KUKA KRL program: cuadrado.src, cuadrado.dat

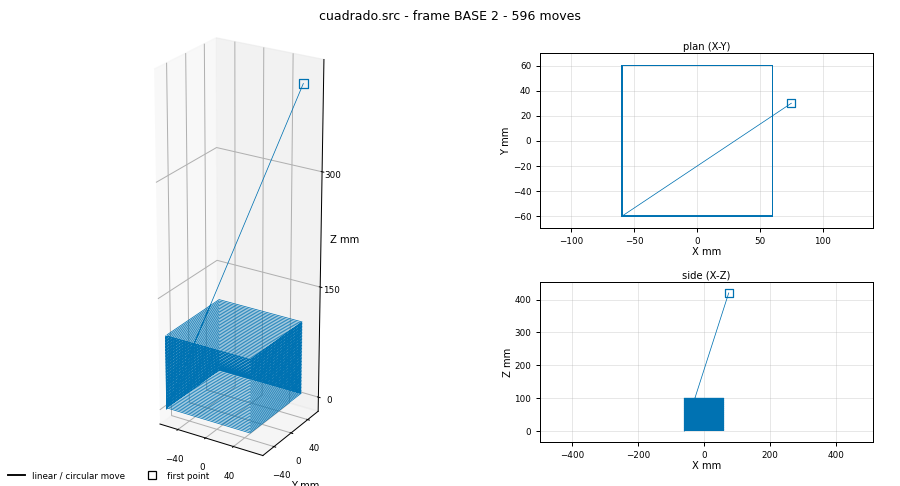
[picture p0: tool path of cuadrado.src in frame BASE 2, 596 of 598 moves have a stored position in this frame; points joined in program order, loops and branches not executed]
--- cuadrado.src ---
&ACCESS RVP
&PARAM TEMPLATE = C:\KRC\Roboter\Template\vorgabe
&PARAM EDITMASK = *
DEF cuadrado( )
;FOLD INI;%{PE}%V3.2.0,%MKUKATPBASIS,%CINIT,%VCOMMON,%P
;FOLD BAS INI;%{E}%V3.2.0,%MKUKATPBASIS,%CINIT,%VINIT,%P
GLOBAL INTERRUPT DECL 3 WHEN $STOPMESS==TRUE DO IR_STOPM ( )
INTERRUPT ON 3
BAS (#INITMOV,0 )
;ENDFOLD (BAS INI)
;FOLD A20 INI;%{E}%V3.2.0,%MKUKATPA20,%CINIT,%VINIT,%P
IF ARC20==TRUE THEN
A20 (ARC_INI)
INTERRUPT DECL 6 WHEN $CYCFLAG[3]==FALSE DO A20(TECH_STOP2)
ENDIF
;ENDFOLD (A20 INI)
;FOLD A10 INI;%{E}%V3.2.0,%MKUKATPARC,%CINIT,%VINIT,%P
IF A10_OPTION==#ACTIVE THEN
INTERRUPT DECL 4 WHEN $CYCFLAG[2]==FALSE DO A10 (#APPL_ERROR)
INTERRUPT DECL 7 WHEN A_ARC_SWI==#ACTIVE DO A10 (#ARC_SEAM)
INTERRUPT DECL 5 WHEN A_FLY_ARC==TRUE DO A10 (#HPU_ARC)
INTERRUPT  ON 5
A10_INI ( )
ENDIF
;ENDFOLD (A10 INI)
;FOLD GRIPPER INI;%{E}%V3.2.0,%MKUKATPGRIPPER,%CINIT,%VINIT,%P
USER_GRP(0,DUMMY,DUMMY,GDEFAULT)
;ENDFOLD (GRIPPER INI)
;FOLD SPOT INI;%{E}%V3.2.0,%MKUKATPSPOT,%CINIT,%VINIT,%P
USERSPOT(#INIT)
;ENDFOLD (SPOT INI)
;FOLD TOUCHSENSE INI;%{E}%V3.2.0,%MKUKATPTS,%CINIT,%VINIT,%P
IF H70_OPTION THEN
INTERRUPT DECL 15 WHEN $MEAS_PULSE[TOUCH_I[TOUCH_ACTIVE].IN_NR] DO H70 (6,CD0 )
INTERRUPT DECL 16 WHEN $ZERO_MOVE DO H70 (7,CD0 )
INTERRUPT DECL 17 WHEN $TECHPAR_C[FG_TOUCH,8]>0.5 DO H70 (8,CD0)
H70 (1,CD0 )
ENDIF
;ENDFOLD (TOUCHSENSE INI)
;FOLD USER INI;%{E}%V3.2.0,%MKUKATPUSER,%CINIT,%VINIT,%P
;Make your modifications here
;ENDFOLD (USER INI)
;ENDFOLD (INI)
; SPEED PTP FOR AXIS
$VEL_AXIS[1] = 15
$VEL_AXIS[2] = 15
$VEL_AXIS[3] = 15
$VEL_AXIS[4] = 15
$VEL_AXIS[5] = 15
$VEL_AXIS[6] = 15
;SMOOTHNESS
$APO.CDIS = 2
;ADVANCE
$ADVANCE = 3
;SET TOOL AND BASE
$TOOL = TOOL_DATA[3]
$BASE = BASE_DATA[2]
;HOME
;FOLD PTP HOME Vel=10% DEFAULT
$BWDSTART=FALSE
$H_POS=XHOME
PDAT_ACT=PDEFAULT
FDAT_ACT=FHOME
BAS(#PTP_DAT )
BAS (#VEL_PTP,10 )
PTP XHOME
;ENDFOLD
;USER PROGRAM
;SPEED $VEL.CP
$VEL.CP=0.025
; OUT[TEMP] = 200
; OUT[vent] = 1
; OUT[RPM] = 25
$OUT[1] = TRUE
WAIT SEC 20
$OUT[1] = FALSE
; USER POSES CALLS
PTP {X 75, Y 30, Z 420, A 0, B 90, C 0}
; USER POSES CALLS
LIN {X -60.0, Y -60.0, Z 0.0, A 0, B 90, C 0} C_DIS
WAIT SEC 3
LIN {X -60.0, Y -60.0, Z 2.0, A 0, B 90, C 0} C_DIS
$OUT[1] = TRUE
WAIT SEC 0.8
LIN {X -60.0, Y -60.0, Z 2.0, A 0, B 90, C 0} C_DIS
LIN {X -60.0, Y -60.0, Z 2.0, A 0, B 90, C 0} C_DIS
LIN {X 60.0, Y -60.0, Z 2.0, A 0, B 90, C 0} C_DIS
LIN {X 60.0, Y 60.0, Z 2.0, A 0, B 90, C 0} C_DIS
LIN {X -60.0, Y 60.0, Z 2.0, A 0, B 90, C 0} C_DIS
LIN {X -60.0, Y -56.5, Z 2.0, A 0, B 90, C 0} C_DIS
$OUT[1] = FALSE

; END LAYER 0
LIN {X -60.0, Y -60.0, Z 2.0, A 0, B 90, C 0} C_DIS
WAIT SEC 3
LIN {X -60.0, Y -60.0, Z 4.0, A 0, B 90, C 0} C_DIS
$OUT[1] = TRUE
WAIT SEC 0.8
LIN {X -60.0, Y -60.0, Z 4.0, A 0, B 90, C 0} C_DIS
LIN {X -60.0, Y -60.0, Z 4.0, A 0, B 90, C 0} C_DIS
LIN {X 57.6, Y -60.0, Z 4.0, A 0, B 90, C 0} C_DIS
LIN {X 60.0, Y -60.0, Z 4.0, A 0, B 90, C 0} C_DIS
LIN {X 60.0, Y 57.6, Z 4.0, A 0, B 90, C 0} C_DIS
LIN {X 60.0, Y 60.0, Z 4.0, A 0, B 90, C 0} C_DIS
LIN {X -57.6, Y 60.0, Z 4.0, A 0, B 90, C 0} C_DIS
LIN {X -60.0, Y 60.0, Z 4.0, A 0, B 90, C 0} C_DIS
LIN {X -60.0, Y -57.6, Z 4.0, A 0, B 90, C 0} C_DIS
$OUT[1] = FALSE

; END LAYER 1
LIN {X -60.0, Y -60.0, Z 4.0, A 0, B 90, C 0} C_DIS
WAIT SEC 3
LIN {X -60.0, Y -60.0, Z 6.0, A 0, B 90, C 0} C_DIS
$OUT[1] = TRUE
WAIT SEC 0.8
LIN {X -60.0, Y -60.0, Z 6.0, A 0, B 90, C 0} C_DIS
LIN {X -60.0, Y -60.0, Z 6.0, A 0, B 90, C 0} C_DIS
LIN {X 55.2, Y -60.0, Z 6.0, A 0, B 90, C 0} C_DIS
LIN {X 60.0, Y -60.0, Z 6.0, A 0, B 90, C 0} C_DIS
LIN {X 60.0, Y 55.2, Z 6.0, A 0, B 90, C 0} C_DIS
LIN {X 60.0, Y 60.0, Z 6.0, A 0, B 90, C 0} C_DIS
LIN {X -55.2, Y 60.0, Z 6.0, A 0, B 90, C 0} C_DIS
LIN {X -60.0, Y 60.0, Z 6.0, A 0, B 90, C 0} C_DIS
LIN {X -60.0, Y -55.2, Z 6.0, A 0, B 90, C 0} C_DIS
LIN {X -60.0, Y -56.5, Z 6.0, A 0, B 90, C 0} C_DIS
$OUT[1] = FALSE

; END LAYER 2
LIN {X -60.0, Y -60.0, Z 6.0, A 0, B 90, C 0} C_DIS
WAIT SEC 3
LIN {X -60.0, Y -60.0, Z 8.0, A 0, B 90, C 0} C_DIS
$OUT[1] = TRUE
WAIT SEC 0.8
LIN {X -60.0, Y -60.0, Z 8.0, A 0, B 90, C 0} C_DIS
LIN {X -60.0, Y -60.0, Z 8.0, A 0, B 90, C 0} C_DIS
LIN {X 52.8, Y -60.0, Z 8.0, A 0, B 90, C 0} C_DIS
LIN {X 60.0, Y -60.0, Z 8.0, A 0, B 90, C 0} C_DIS
LIN {X 60.0, Y 52.8, Z 8.0, A 0, B 90, C 0} C_DIS
LIN {X 60.0, Y 60.0, Z 8.0, A 0, B 90, C 0} C_DIS
LIN {X -52.8, Y 60.0, Z 8.0, A 0, B 90, C 0} C_DIS
LIN {X -60.0, Y 60.0, Z 8.0, A 0, B 90, C 0} C_DIS
LIN {X -60.0, Y -52.8, Z 8.0, A 0, B 90, C 0} C_DIS
LIN {X -60.0, Y -56.5, Z 8.0, A 0, B 90, C 0} C_DIS
$OUT[1] = FALSE

; END LAYER 3
LIN {X -60.0, Y -60.0, Z 8.0, A 0, B 90, C 0} C_DIS
WAIT SEC 3
LIN {X -60.0, Y -60.0, Z 10.0, A 0, B 90, C 0} C_DIS
$OUT[1] = TRUE
WAIT SEC 0.8
LIN {X -60.0, Y -60.0, Z 10.0, A 0, B 90, C 0} C_DIS
LIN {X -60.0, Y -60.0, Z 10.0, A 0, B 90, C 0} C_DIS
LIN {X 50.4, Y -60.0, Z 10.0, A 0, B 90, C 0} C_DIS
LIN {X 60.0, Y -60.0, Z 10.0, A 0, B 90, C 0} C_DIS
LIN {X 60.0, Y 50.4, Z 10.0, A 0, B 90, C 0} C_DIS
LIN {X 60.0, Y 60.0, Z 10.0, A 0, B 90, C 0} C_DIS
LIN {X -50.4, Y 60.0, Z 10.0, A 0, B 90, C 0} C_DIS
LIN {X -60.0, Y 60.0, Z 10.0, A 0, B 90, C 0} C_DIS
LIN {X -60.0, Y -50.4, Z 10.0, A 0, B 90, C 0} C_DIS
LIN {X -60.0, Y -56.5, Z 10.0, A 0, B 90, C 0} C_DIS
$OUT[1] = FALSE

; END LAYER 4
LIN {X -60.0, Y -60.0, Z 10.0, A 0, B 90, C 0} C_DIS
WAIT SEC 3
LIN {X -60.0, Y -60.0, Z 12.0, A 0, B 90, C 0} C_DIS
$OUT[1] = TRUE
WAIT SEC 0.8
LIN {X -60.0, Y -60.0, Z 12.0, A 0, B 90, C 0} C_DIS
LIN {X -60.0, Y -60.0, Z 12.0, A 0, B 90, C 0} C_DIS
LIN {X 48.0, Y -60.0, Z 12.0, A 0, B 90, C 0} C_DIS
LIN {X 60.0, Y -60.0, Z 12.0, A 0, B 90, C 0} C_DIS
LIN {X 60.0, Y 48.0, Z 12.0, A 0, B 90, C 0} C_DIS
LIN {X 60.0, Y 60.0, Z 12.0, A 0, B 90, C 0} C_DIS
LIN {X -48.0, Y 60.0, Z 12.0, A 0, B 90, C 0} C_DIS
LIN {X -60.0, Y 60.0, Z 12.0, A 0, B 90, C 0} C_DIS
LIN {X -60.0, Y -48.0, Z 12.0, A 0, B 90, C 0} C_DIS
LIN {X -60.0, Y -56.5, Z 12.0, A 0, B 90, C 0} C_DIS
$OUT[1] = FALSE

; END LAYER 5
LIN {X -60.0, Y -60.0, Z 12.0, A 0, B 90, C 0} C_DIS
WAIT SEC 3
LIN {X -60.0, Y -60.0, Z 14.0, A 0, B 90, C 0} C_DIS
$OUT[1] = TRUE
WAIT SEC 0.8
LIN {X -60.0, Y -60.0, Z 14.0, A 0, B 90, C 0} C_DIS
LIN {X -60.0, Y -60.0, Z 14.0, A 0, B 90, C 0} C_DIS
LIN {X 45.6, Y -60.0, Z 14.0, A 0, B 90, C 0} C_DIS
LIN {X 60.0, Y -60.0, Z 14.0, A 0, B 90, C 0} C_DIS
LIN {X 60.0, Y 45.6, Z 14.0, A 0, B 90, C 0} C_DIS
LIN {X 60.0, Y 60.0, Z 14.0, A 0, B 90, C 0} C_DIS
LIN {X -45.6, Y 60.0, Z 14.0, A 0, B 90, C 0} C_DIS
LIN {X -60.0, Y 60.0, Z 14.0, A 0, B 90, C 0} C_DIS
LIN {X -60.0, Y -45.6, Z 14.0, A 0, B 90, C 0} C_DIS
LIN {X -60.0, Y -56.5, Z 14.0, A 0, B 90, C 0} C_DIS
$OUT[1] = FALSE

; END LAYER 6
LIN {X -60.0, Y -60.0, Z 14.0, A 0, B 90, C 0} C_DIS
WAIT SEC 3
LIN {X -60.0, Y -60.0, Z 16.0, A 0, B 90, C 0} C_DIS
$OUT[1] = TRUE
WAIT SEC 0.8
LIN {X -60.0, Y -60.0, Z 16.0, A 0, B 90, C 0} C_DIS
LIN {X -60.0, Y -60.0, Z 16.0, A 0, B 90, C 0} C_DIS
LIN {X 43.2, Y -60.0, Z 16.0, A 0, B 90, C 0} C_DIS
LIN {X 60.0, Y -60.0, Z 16.0, A 0, B 90, C 0} C_DIS
LIN {X 60.0, Y 43.2, Z 16.0, A 0, B 90, C 0} C_DIS
LIN {X 60.0, Y 60.0, Z 16.0, A 0, B 90, C 0} C_DIS
LIN {X -43.2, Y 60.0, Z 16.0, A 0, B 90, C 0} C_DIS
LIN {X -60.0, Y 60.0, Z 16.0, A 0, B 90, C 0} C_DIS
LIN {X -60.0, Y -43.2, Z 16.0, A 0, B 90, C 0} C_DIS
LIN {X -60.0, Y -56.5, Z 16.0, A 0, B 90, C 0} C_DIS
$OUT[1] = FALSE

; END LAYER 7
LIN {X -60.0, Y -60.0, Z 16.0, A 0, B 90, C 0} C_DIS
WAIT SEC 3
LIN {X -60.0, Y -60.0, Z 18.0, A 0, B 90, C 0} C_DIS
$OUT[1] = TRUE
WAIT SEC 0.8
LIN {X -60.0, Y -60.0, Z 18.0, A 0, B 90, C 0} C_DIS
LIN {X -60.0, Y -60.0, Z 18.0, A 0, B 90, C 0} C_DIS
LIN {X 40.8, Y -60.0, Z 18.0, A 0, B 90, C 0} C_DIS
LIN {X 60.0, Y -60.0, Z 18.0, A 0, B 90, C 0} C_DIS
LIN {X 60.0, Y 40.8, Z 18.0, A 0, B 90, C 0} C_DIS
LIN {X 60.0, Y 60.0, Z 18.0, A 0, B 90, C 0} C_DIS
LIN {X -40.8, Y 60.0, Z 18.0, A 0, B 90, C 0} C_DIS
LIN {X -60.0, Y 60.0, Z 18.0, A 0, B 90, C 0} C_DIS
LIN {X -60.0, Y -40.8, Z 18.0, A 0, B 90, C 0} C_DIS
LIN {X -60.0, Y -56.5, Z 18.0, A 0, B 90, C 0} C_DIS
$OUT[1] = FALSE

; END LAYER 8
LIN {X -60.0, Y -60.0, Z 18.0, A 0, B 90, C 0} C_DIS
WAIT SEC 3
LIN {X -60.0, Y -60.0, Z 20.0, A 0, B 90, C 0} C_DIS
$OUT[1] = TRUE
WAIT SEC 0.8
LIN {X -60.0, Y -60.0, Z 20.0, A 0, B 90, C 0} C_DIS
LIN {X -60.0, Y -60.0, Z 20.0, A 0, B 90, C 0} C_DIS
LIN {X 38.4, Y -60.0, Z 20.0, A 0, B 90, C 0} C_DIS
LIN {X 60.0, Y -60.0, Z 20.0, A 0, B 90, C 0} C_DIS
LIN {X 60.0, Y 38.4, Z 20.0, A 0, B 90, C 0} C_DIS
LIN {X 60.0, Y 60.0, Z 20.0, A 0, B 90, C 0} C_DIS
LIN {X -38.4, Y 60.0, Z 20.0, A 0, B 90, C 0} C_DIS
LIN {X -60.0, Y 60.0, Z 20.0, A 0, B 90, C 0} C_DIS
LIN {X -60.0, Y -38.4, Z 20.0, A 0, B 90, C 0} C_DIS
LIN {X -60.0, Y -56.5, Z 20.0, A 0, B 90, C 0} C_DIS
$OUT[1] = FALSE

; END LAYER 9
LIN {X -60.0, Y -60.0, Z 20.0, A 0, B 90, C 0} C_DIS
WAIT SEC 3
LIN {X -60.0, Y -60.0, Z 22.0, A 0, B 90, C 0} C_DIS
$OUT[1] = TRUE
WAIT SEC 0.8
LIN {X -60.0, Y -60.0, Z 22.0, A 0, B 90, C 0} C_DIS
LIN {X -60.0, Y -60.0, Z 22.0, A 0, B 90, C 0} C_DIS
LIN {X 36.0, Y -60.0, Z 22.0, A 0, B 90, C 0} C_DIS
LIN {X 60.0, Y -60.0, Z 22.0, A 0, B 90, C 0} C_DIS
LIN {X 60.0, Y 36.0, Z 22.0, A 0, B 90, C 0} C_DIS
LIN {X 60.0, Y 60.0, Z 22.0, A 0, B 90, C 0} C_DIS
LIN {X -36.0, Y 60.0, Z 22.0, A 0, B 90, C 0} C_DIS
LIN {X -60.0, Y 60.0, Z 22.0, A 0, B 90, C 0} C_DIS
LIN {X -60.0, Y -36.0, Z 22.0, A 0, B 90, C 0} C_DIS
LIN {X -60.0, Y -56.5, Z 22.0, A 0, B 90, C 0} C_DIS
$OUT[1] = FALSE

; END LAYER 10
LIN {X -60.0, Y -60.0, Z 22.0, A 0, B 90, C 0} C_DIS
WAIT SEC 3
LIN {X -60.0, Y -60.0, Z 24.0, A 0, B 90, C 0} C_DIS
$OUT[1] = TRUE
WAIT SEC 0.8
LIN {X -60.0, Y -60.0, Z 24.0, A 0, B 90, C 0} C_DIS
LIN {X -60.0, Y -60.0, Z 24.0, A 0, B 90, C 0} C_DIS
LIN {X 33.6, Y -60.0, Z 24.0, A 0, B 90, C 0} C_DIS
LIN {X 60.0, Y -60.0, Z 24.0, A 0, B 90, C 0} C_DIS
LIN {X 60.0, Y 33.6, Z 24.0, A 0, B 90, C 0} C_DIS
LIN {X 60.0, Y 60.0, Z 24.0, A 0, B 90, C 0} C_DIS
LIN {X -33.6, Y 60.0, Z 24.0, A 0, B 90, C 0} C_DIS
LIN {X -60.0, Y 60.0, Z 24.0, A 0, B 90, C 0} C_DIS
LIN {X -60.0, Y -33.6, Z 24.0, A 0, B 90, C 0} C_DIS
LIN {X -60.0, Y -56.5, Z 24.0, A 0, B 90, C 0} C_DIS
$OUT[1] = FALSE

; END LAYER 11
LIN {X -60.0, Y -60.0, Z 24.0, A 0, B 90, C 0} C_DIS
WAIT SEC 3
LIN {X -60.0, Y -60.0, Z 26.0, A 0, B 90, C 0} C_DIS
$OUT[1] = TRUE
WAIT SEC 0.8
LIN {X -60.0, Y -60.0, Z 26.0, A 0, B 90, C 0} C_DIS
LIN {X -60.0, Y -60.0, Z 26.0, A 0, B 90, C 0} C_DIS
LIN {X 31.2, Y -60.0, Z 26.0, A 0, B 90, C 0} C_DIS
LIN {X 60.0, Y -60.0, Z 26.0, A 0, B 90, C 0} C_DIS
LIN {X 60.0, Y 31.2, Z 26.0, A 0, B 90, C 0} C_DIS
LIN {X 60.0, Y 60.0, Z 26.0, A 0, B 90, C 0} C_DIS
LIN {X -31.2, Y 60.0, Z 26.0, A 0, B 90, C 0} C_DIS
LIN {X -60.0, Y 60.0, Z 26.0, A 0, B 90, C 0} C_DIS
LIN {X -60.0, Y -31.2, Z 26.0, A 0, B 90, C 0} C_DIS
LIN {X -60.0, Y -56.5, Z 26.0, A 0, B 90, C 0} C_DIS
$OUT[1] = FALSE

; END LAYER 12
LIN {X -60.0, Y -60.0, Z 26.0, A 0, B 90, C 0} C_DIS
WAIT SEC 3
LIN {X -60.0, Y -60.0, Z 28.0, A 0, B 90, C 0} C_DIS
$OUT[1] = TRUE
WAIT SEC 0.8
LIN {X -60.0, Y -60.0, Z 28.0, A 0, B 90, C 0} C_DIS
LIN {X -60.0, Y -60.0, Z 28.0, A 0, B 90, C 0} C_DIS
LIN {X 28.8, Y -60.0, Z 28.0, A 0, B 90, C 0} C_DIS
LIN {X 60.0, Y -60.0, Z 28.0, A 0, B 90, C 0} C_DIS
LIN {X 60.0, Y 28.8, Z 28.0, A 0, B 90, C 0} C_DIS
LIN {X 60.0, Y 60.0, Z 28.0, A 0, B 90, C 0} C_DIS
LIN {X -28.8, Y 60.0, Z 28.0, A 0, B 90, C 0} C_DIS
LIN {X -60.0, Y 60.0, Z 28.0, A 0, B 90, C 0} C_DIS
LIN {X -60.0, Y -28.8, Z 28.0, A 0, B 90, C 0} C_DIS
LIN {X -60.0, Y -56.5, Z 28.0, A 0, B 90, C 0} C_DIS
$OUT[1] = FALSE

; END LAYER 13
LIN {X -60.0, Y -60.0, Z 28.0, A 0, B 90, C 0} C_DIS
WAIT SEC 3
LIN {X -60.0, Y -60.0, Z 30.0, A 0, B 90, C 0} C_DIS
$OUT[1] = TRUE
WAIT SEC 0.8
LIN {X -60.0, Y -60.0, Z 30.0, A 0, B 90, C 0} C_DIS
LIN {X -60.0, Y -60.0, Z 30.0, A 0, B 90, C 0} C_DIS
LIN {X 26.4, Y -60.0, Z 30.0, A 0, B 90, C 0} C_DIS
LIN {X 60.0, Y -60.0, Z 30.0, A 0, B 90, C 0} C_DIS
LIN {X 60.0, Y 26.4, Z 30.0, A 0, B 90, C 0} C_DIS
LIN {X 60.0, Y 60.0, Z 30.0, A 0, B 90, C 0} C_DIS
LIN {X -26.4, Y 60.0, Z 30.0, A 0, B 90, C 0} C_DIS
LIN {X -60.0, Y 60.0, Z 30.0, A 0, B 90, C 0} C_DIS
LIN {X -60.0, Y -26.4, Z 30.0, A 0, B 90, C 0} C_DIS
LIN {X -60.0, Y -56.5, Z 30.0, A 0, B 90, C 0} C_DIS
$OUT[1] = FALSE

; END LAYER 14
LIN {X -60.0, Y -60.0, Z 30.0, A 0, B 90, C 0} C_DIS
WAIT SEC 3
LIN {X -60.0, Y -60.0, Z 32.0, A 0, B 90, C 0} C_DIS
$OUT[1] = TRUE
WAIT SEC 0.8
LIN {X -60.0, Y -60.0, Z 32.0, A 0, B 90, C 0} C_DIS
LIN {X -60.0, Y -60.0, Z 32.0, A 0, B 90, C 0} C_DIS
LIN {X 24.0, Y -60.0, Z 32.0, A 0, B 90, C 0} C_DIS
LIN {X 60.0, Y -60.0, Z 32.0, A 0, B 90, C 0} C_DIS
LIN {X 60.0, Y 24.0, Z 32.0, A 0, B 90, C 0} C_DIS
LIN {X 60.0, Y 60.0, Z 32.0, A 0, B 90, C 0} C_DIS
LIN {X -24.0, Y 60.0, Z 32.0, A 0, B 90, C 0} C_DIS
LIN {X -60.0, Y 60.0, Z 32.0, A 0, B 90, C 0} C_DIS
LIN {X -60.0, Y -24.0, Z 32.0, A 0, B 90, C 0} C_DIS
LIN {X -60.0, Y -56.5, Z 32.0, A 0, B 90, C 0} C_DIS
$OUT[1] = FALSE

; END LAYER 15
LIN {X -60.0, Y -60.0, Z 32.0, A 0, B 90, C 0} C_DIS
WAIT SEC 3
LIN {X -60.0, Y -60.0, Z 34.0, A 0, B 90, C 0} C_DIS
$OUT[1] = TRUE
WAIT SEC 0.8
LIN {X -60.0, Y -60.0, Z 34.0, A 0, B 90, C 0} C_DIS
LIN {X -60.0, Y -60.0, Z 34.0, A 0, B 90, C 0} C_DIS
LIN {X 21.6, Y -60.0, Z 34.0, A 0, B 90, C 0} C_DIS
LIN {X 60.0, Y -60.0, Z 34.0, A 0, B 90, C 0} C_DIS
LIN {X 60.0, Y 21.6, Z 34.0, A 0, B 90, C 0} C_DIS
LIN {X 60.0, Y 60.0, Z 34.0, A 0, B 90, C 0} C_DIS
LIN {X -21.6, Y 60.0, Z 34.0, A 0, B 90, C 0} C_DIS
LIN {X -60.0, Y 60.0, Z 34.0, A 0, B 90, C 0} C_DIS
LIN {X -60.0, Y -21.6, Z 34.0, A 0, B 90, C 0} C_DIS
LIN {X -60.0, Y -56.5, Z 34.0, A 0, B 90, C 0} C_DIS
$OUT[1] = FALSE

; END LAYER 16
LIN {X -60.0, Y -60.0, Z 34.0, A 0, B 90, C 0} C_DIS
WAIT SEC 3
LIN {X -60.0, Y -60.0, Z 36.0, A 0, B 90, C 0} C_DIS
$OUT[1] = TRUE
WAIT SEC 0.8
LIN {X -60.0, Y -60.0, Z 36.0, A 0, B 90, C 0} C_DIS
LIN {X -60.0, Y -60.0, Z 36.0, A 0, B 90, C 0} C_DIS
LIN {X 19.2, Y -60.0, Z 36.0, A 0, B 90, C 0} C_DIS
LIN {X 60.0, Y -60.0, Z 36.0, A 0, B 90, C 0} C_DIS
LIN {X 60.0, Y 19.2, Z 36.0, A 0, B 90, C 0} C_DIS
LIN {X 60.0, Y 60.0, Z 36.0, A 0, B 90, C 0} C_DIS
LIN {X -19.2, Y 60.0, Z 36.0, A 0, B 90, C 0} C_DIS
LIN {X -60.0, Y 60.0, Z 36.0, A 0, B 90, C 0} C_DIS
LIN {X -60.0, Y -19.2, Z 36.0, A 0, B 90, C 0} C_DIS
LIN {X -60.0, Y -56.5, Z 36.0, A 0, B 90, C 0} C_DIS
$OUT[1] = FALSE

; END LAYER 17
LIN {X -60.0, Y -60.0, Z 36.0, A 0, B 90, C 0} C_DIS
WAIT SEC 3
LIN {X -60.0, Y -60.0, Z 38.0, A 0, B 90, C 0} C_DIS
$OUT[1] = TRUE
WAIT SEC 0.8
LIN {X -60.0, Y -60.0, Z 38.0, A 0, B 90, C 0} C_DIS
LIN {X -60.0, Y -60.0, Z 38.0, A 0, B 90, C 0} C_DIS
LIN {X 16.8, Y -60.0, Z 38.0, A 0, B 90, C 0} C_DIS
LIN {X 60.0, Y -60.0, Z 38.0, A 0, B 90, C 0} C_DIS
LIN {X 60.0, Y 16.8, Z 38.0, A 0, B 90, C 0} C_DIS
LIN {X 60.0, Y 60.0, Z 38.0, A 0, B 90, C 0} C_DIS
LIN {X -16.8, Y 60.0, Z 38.0, A 0, B 90, C 0} C_DIS
LIN {X -60.0, Y 60.0, Z 38.0, A 0, B 90, C 0} C_DIS
LIN {X -60.0, Y -16.8, Z 38.0, A 0, B 90, C 0} C_DIS
LIN {X -60.0, Y -56.5, Z 38.0, A 0, B 90, C 0} C_DIS
$OUT[1] = FALSE

; END LAYER 18
LIN {X -60.0, Y -60.0, Z 38.0, A 0, B 90, C 0} C_DIS
WAIT SEC 3
LIN {X -60.0, Y -60.0, Z 40.0, A 0, B 90, C 0} C_DIS
$OUT[1] = TRUE
WAIT SEC 0.8
LIN {X -60.0, Y -60.0, Z 40.0, A 0, B 90, C 0} C_DIS
LIN {X -60.0, Y -60.0, Z 40.0, A 0, B 90, C 0} C_DIS
LIN {X 14.4, Y -60.0, Z 40.0, A 0, B 90, C 0} C_DIS
LIN {X 60.0, Y -60.0, Z 40.0, A 0, B 90, C 0} C_DIS
LIN {X 60.0, Y 14.4, Z 40.0, A 0, B 90, C 0} C_DIS
LIN {X 60.0, Y 60.0, Z 40.0, A 0, B 90, C 0} C_DIS
LIN {X -14.4, Y 60.0, Z 40.0, A 0, B 90, C 0} C_DIS
LIN {X -60.0, Y 60.0, Z 40.0, A 0, B 90, C 0} C_DIS
LIN {X -60.0, Y -14.4, Z 40.0, A 0, B 90, C 0} C_DIS
LIN {X -60.0, Y -56.5, Z 40.0, A 0, B 90, C 0} C_DIS
$OUT[1] = FALSE

; END LAYER 19
LIN {X -60.0, Y -60.0, Z 40.0, A 0, B 90, C 0} C_DIS
WAIT SEC 3
LIN {X -60.0, Y -60.0, Z 42.0, A 0, B 90, C 0} C_DIS
$OUT[1] = TRUE
WAIT SEC 0.8
LIN {X -60.0, Y -60.0, Z 42.0, A 0, B 90, C 0} C_DIS
LIN {X -60.0, Y -60.0, Z 42.0, A 0, B 90, C 0} C_DIS
LIN {X 12.0, Y -60.0, Z 42.0, A 0, B 90, C 0} C_DIS
LIN {X 60.0, Y -60.0, Z 42.0, A 0, B 90, C 0} C_DIS
LIN {X 60.0, Y 12.0, Z 42.0, A 0, B 90, C 0} C_DIS
LIN {X 60.0, Y 60.0, Z 42.0, A 0, B 90, C 0} C_DIS
LIN {X -12.0, Y 60.0, Z 42.0, A 0, B 90, C 0} C_DIS
LIN {X -60.0, Y 60.0, Z 42.0, A 0, B 90, C 0} C_DIS
LIN {X -60.0, Y -12.0, Z 42.0, A 0, B 90, C 0} C_DIS
LIN {X -60.0, Y -56.5, Z 42.0, A 0, B 90, C 0} C_DIS
$OUT[1] = FALSE

; END LAYER 20
LIN {X -60.0, Y -60.0, Z 42.0, A 0, B 90, C 0} C_DIS
WAIT SEC 3
LIN {X -60.0, Y -60.0, Z 44.0, A 0, B 90, C 0} C_DIS
$OUT[1] = TRUE
WAIT SEC 0.8
LIN {X -60.0, Y -60.0, Z 44.0, A 0, B 90, C 0} C_DIS
LIN {X -60.0, Y -60.0, Z 44.0, A 0, B 90, C 0} C_DIS
LIN {X 9.6, Y -60.0, Z 44.0, A 0, B 90, C 0} C_DIS
LIN {X 60.0, Y -60.0, Z 44.0, A 0, B 90, C 0} C_DIS
LIN {X 60.0, Y 9.6, Z 44.0, A 0, B 90, C 0} C_DIS
LIN {X 60.0, Y 60.0, Z 44.0, A 0, B 90, C 0} C_DIS
LIN {X -9.6, Y 60.0, Z 44.0, A 0, B 90, C 0} C_DIS
LIN {X -60.0, Y 60.0, Z 44.0, A 0, B 90, C 0} C_DIS
LIN {X -60.0, Y -9.6, Z 44.0, A 0, B 90, C 0} C_DIS
LIN {X -60.0, Y -56.5, Z 44.0, A 0, B 90, C 0} C_DIS
$OUT[1] = FALSE

; END LAYER 21
LIN {X -60.0, Y -60.0, Z 44.0, A 0, B 90, C 0} C_DIS
WAIT SEC 3
LIN {X -60.0, Y -60.0, Z 46.0, A 0, B 90, C 0} C_DIS
$OUT[1] = TRUE
WAIT SEC 0.8
LIN {X -60.0, Y -60.0, Z 46.0, A 0, B 90, C 0} C_DIS
LIN {X -60.0, Y -60.0, Z 46.0, A 0, B 90, C 0} C_DIS
LIN {X 7.2, Y -60.0, Z 46.0, A 0, B 90, C 0} C_DIS
LIN {X 60.0, Y -60.0, Z 46.0, A 0, B 90, C 0} C_DIS
LIN {X 60.0, Y 7.2, Z 46.0, A 0, B 90, C 0} C_DIS
LIN {X 60.0, Y 60.0, Z 46.0, A 0, B 90, C 0} C_DIS
LIN {X -7.2, Y 60.0, Z 46.0, A 0, B 90, C 0} C_DIS
LIN {X -60.0, Y 60.0, Z 46.0, A 0, B 90, C 0} C_DIS
LIN {X -60.0, Y -7.2, Z 46.0, A 0, B 90, C 0} C_DIS
LIN {X -60.0, Y -56.5, Z 46.0, A 0, B 90, C 0} C_DIS
$OUT[1] = FALSE

; END LAYER 22
LIN {X -60.0, Y -60.0, Z 46.0, A 0, B 90, C 0} C_DIS
WAIT SEC 3
LIN {X -60.0, Y -60.0, Z 48.0, A 0, B 90, C 0} C_DIS
$OUT[1] = TRUE
WAIT SEC 0.8
LIN {X -60.0, Y -60.0, Z 48.0, A 0, B 90, C 0} C_DIS
LIN {X -60.0, Y -60.0, Z 48.0, A 0, B 90, C 0} C_DIS
LIN {X 4.8, Y -60.0, Z 48.0, A 0, B 90, C 0} C_DIS
LIN {X 60.0, Y -60.0, Z 48.0, A 0, B 90, C 0} C_DIS
LIN {X 60.0, Y 4.8, Z 48.0, A 0, B 90, C 0} C_DIS
LIN {X 60.0, Y 60.0, Z 48.0, A 0, B 90, C 0} C_DIS
LIN {X -4.8, Y 60.0, Z 48.0, A 0, B 90, C 0} C_DIS
LIN {X -60.0, Y 60.0, Z 48.0, A 0, B 90, C 0} C_DIS
LIN {X -60.0, Y -4.8, Z 48.0, A 0, B 90, C 0} C_DIS
LIN {X -60.0, Y -56.5, Z 48.0, A 0, B 90, C 0} C_DIS
$OUT[1] = FALSE

; END LAYER 23
LIN {X -60.0, Y -60.0, Z 48.0, A 0, B 90, C 0} C_DIS
WAIT SEC 3
LIN {X -60.0, Y -60.0, Z 50.0, A 0, B 90, C 0} C_DIS
$OUT[1] = TRUE
WAIT SEC 0.8
LIN {X -60.0, Y -60.0, Z 50.0, A 0, B 90, C 0} C_DIS
LIN {X -60.0, Y -60.0, Z 50.0, A 0, B 90, C 0} C_DIS
LIN {X 2.4, Y -60.0, Z 50.0, A 0, B 90, C 0} C_DIS
LIN {X 60.0, Y -60.0, Z 50.0, A 0, B 90, C 0} C_DIS
LIN {X 60.0, Y 2.4, Z 50.0, A 0, B 90, C 0} C_DIS
LIN {X 60.0, Y 60.0, Z 50.0, A 0, B 90, C 0} C_DIS
LIN {X -2.4, Y 60.0, Z 50.0, A 0, B 90, C 0} C_DIS
LIN {X -60.0, Y 60.0, Z 50.0, A 0, B 90, C 0} C_DIS
LIN {X -60.0, Y -2.4, Z 50.0, A 0, B 90, C 0} C_DIS
LIN {X -60.0, Y -56.5, Z 50.0, A 0, B 90, C 0} C_DIS
$OUT[1] = FALSE

; END LAYER 24
LIN {X -60.0, Y -60.0, Z 50.0, A 0, B 90, C 0} C_DIS
WAIT SEC 3
LIN {X -60.0, Y -60.0, Z 52.0, A 0, B 90, C 0} C_DIS
$OUT[1] = TRUE
WAIT SEC 0.8
LIN {X -60.0, Y -60.0, Z 52.0, A 0, B 90, C 0} C_DIS
LIN {X -60.0, Y -60.0, Z 52.0, A 0, B 90, C 0} C_DIS
LIN {X 0.0, Y -60.0, Z 52.0, A 0, B 90, C 0} C_DIS
LIN {X 60.0, Y -60.0, Z 52.0, A 0, B 90, C 0} C_DIS
LIN {X 60.0, Y 0.0, Z 52.0, A 0, B 90, C 0} C_DIS
LIN {X 60.0, Y 60.0, Z 52.0, A 0, B 90, C 0} C_DIS
LIN {X -0.0, Y 60.0, Z 52.0, A 0, B 90, C 0} C_DIS
LIN {X -60.0, Y 60.0, Z 52.0, A 0, B 90, C 0} C_DIS
LIN {X -60.0, Y -0.0, Z 52.0, A 0, B 90, C 0} C_DIS
LIN {X -60.0, Y -56.5, Z 52.0, A 0, B 90, C 0} C_DIS
$OUT[1] = FALSE

; END LAYER 25
LIN {X -60.0, Y -60.0, Z 52.0, A 0, B 90, C 0} C_DIS
WAIT SEC 3
LIN {X -60.0, Y -60.0, Z 54.0, A 0, B 90, C 0} C_DIS
$OUT[1] = TRUE
WAIT SEC 0.8
LIN {X -60.0, Y -60.0, Z 54.0, A 0, B 90, C 0} C_DIS
LIN {X -60.0, Y -60.0, Z 54.0, A 0, B 90, C 0} C_DIS
LIN {X -2.4, Y -60.0, Z 54.0, A 0, B 90, C 0} C_DIS
LIN {X 60.0, Y -60.0, Z 54.0, A 0, B 90, C 0} C_DIS
LIN {X 60.0, Y -2.4, Z 54.0, A 0, B 90, C 0} C_DIS
LIN {X 60.0, Y 60.0, Z 54.0, A 0, B 90, C 0} C_DIS
LIN {X 2.4, Y 60.0, Z 54.0, A 0, B 90, C 0} C_DIS
LIN {X -60.0, Y 60.0, Z 54.0, A 0, B 90, C 0} C_DIS
LIN {X -60.0, Y 2.4, Z 54.0, A 0, B 90, C 0} C_DIS
LIN {X -60.0, Y -56.5, Z 54.0, A 0, B 90, C 0} C_DIS
$OUT[1] = FALSE

; END LAYER 26
LIN {X -60.0, Y -60.0, Z 54.0, A 0, B 90, C 0} C_DIS
WAIT SEC 3
LIN {X -60.0, Y -60.0, Z 56.0, A 0, B 90, C 0} C_DIS
$OUT[1] = TRUE
WAIT SEC 0.8
LIN {X -60.0, Y -60.0, Z 56.0, A 0, B 90, C 0} C_DIS
LIN {X -60.0, Y -60.0, Z 56.0, A 0, B 90, C 0} C_DIS
LIN {X -4.8, Y -60.0, Z 56.0, A 0, B 90, C 0} C_DIS
LIN {X 60.0, Y -60.0, Z 56.0, A 0, B 90, C 0} C_DIS
LIN {X 60.0, Y -4.8, Z 56.0, A 0, B 90, C 0} C_DIS
LIN {X 60.0, Y 60.0, Z 56.0, A 0, B 90, C 0} C_DIS
LIN {X 4.8, Y 60.0, Z 56.0, A 0, B 90, C 0} C_DIS
LIN {X -60.0, Y 60.0, Z 56.0, A 0, B 90, C 0} C_DIS
LIN {X -60.0, Y 4.8, Z 56.0, A 0, B 90, C 0} C_DIS
LIN {X -60.0, Y -56.5, Z 56.0, A 0, B 90, C 0} C_DIS
$OUT[1] = FALSE

; END LAYER 27
LIN {X -60.0, Y -60.0, Z 56.0, A 0, B 90, C 0} C_DIS
WAIT SEC 3
LIN {X -60.0, Y -60.0, Z 58.0, A 0, B 90, C 0} C_DIS
$OUT[1] = TRUE
WAIT SEC 0.8
LIN {X -60.0, Y -60.0, Z 58.0, A 0, B 90, C 0} C_DIS
LIN {X -60.0, Y -60.0, Z 58.0, A 0, B 90, C 0} C_DIS
LIN {X -7.2, Y -60.0, Z 58.0, A 0, B 90, C 0} C_DIS
LIN {X 60.0, Y -60.0, Z 58.0, A 0, B 90, C 0} C_DIS
LIN {X 60.0, Y -7.2, Z 58.0, A 0, B 90, C 0} C_DIS
LIN {X 60.0, Y 60.0, Z 58.0, A 0, B 90, C 0} C_DIS
LIN {X 7.2, Y 60.0, Z 58.0, A 0, B 90, C 0} C_DIS
LIN {X -60.0, Y 60.0, Z 58.0, A 0, B 90, C 0} C_DIS
LIN {X -60.0, Y 7.2, Z 58.0, A 0, B 90, C 0} C_DIS
LIN {X -60.0, Y -56.5, Z 58.0, A 0, B 90, C 0} C_DIS
$OUT[1] = FALSE

; END LAYER 28
LIN {X -60.0, Y -60.0, Z 58.0, A 0, B 90, C 0} C_DIS
WAIT SEC 3
LIN {X -60.0, Y -60.0, Z 60.0, A 0, B 90, C 0} C_DIS
$OUT[1] = TRUE
WAIT SEC 0.8
LIN {X -60.0, Y -60.0, Z 60.0, A 0, B 90, C 0} C_DIS
LIN {X -60.0, Y -60.0, Z 60.0, A 0, B 90, C 0} C_DIS
LIN {X -9.6, Y -60.0, Z 60.0, A 0, B 90, C 0} C_DIS
LIN {X 60.0, Y -60.0, Z 60.0, A 0, B 90, C 0} C_DIS
LIN {X 60.0, Y -9.6, Z 60.0, A 0, B 90, C 0} C_DIS
LIN {X 60.0, Y 60.0, Z 60.0, A 0, B 90, C 0} C_DIS
LIN {X 9.6, Y 60.0, Z 60.0, A 0, B 90, C 0} C_DIS
LIN {X -60.0, Y 60.0, Z 60.0, A 0, B 90, C 0} C_DIS
LIN {X -60.0, Y 9.6, Z 60.0, A 0, B 90, C 0} C_DIS
LIN {X -60.0, Y -56.5, Z 60.0, A 0, B 90, C 0} C_DIS
$OUT[1] = FALSE

; END LAYER 29
LIN {X -60.0, Y -60.0, Z 60.0, A 0, B 90, C 0} C_DIS
WAIT SEC 3
LIN {X -60.0, Y -60.0, Z 62.0, A 0, B 90, C 0} C_DIS
$OUT[1] = TRUE
WAIT SEC 0.8
LIN {X -60.0, Y -60.0, Z 62.0, A 0, B 90, C 0} C_DIS
LIN {X -60.0, Y -60.0, Z 62.0, A 0, B 90, C 0} C_DIS
LIN {X -12.0, Y -60.0, Z 62.0, A 0, B 90, C 0} C_DIS
LIN {X 60.0, Y -60.0, Z 62.0, A 0, B 90, C 0} C_DIS
LIN {X 60.0, Y -12.0, Z 62.0, A 0, B 90, C 0} C_DIS
LIN {X 60.0, Y 60.0, Z 62.0, A 0, B 90, C 0} C_DIS
LIN {X 12.0, Y 60.0, Z 62.0, A 0, B 90, C 0} C_DIS
LIN {X -60.0, Y 60.0, Z 62.0, A 0, B 90, C 0} C_DIS
LIN {X -60.0, Y 12.0, Z 62.0, A 0, B 90, C 0} C_DIS
LIN {X -60.0, Y -56.5, Z 62.0, A 0, B 90, C 0} C_DIS
$OUT[1] = FALSE

; END LAYER 30
LIN {X -60.0, Y -60.0, Z 62.0, A 0, B 90, C 0} C_DIS
WAIT SEC 3
LIN {X -60.0, Y -60.0, Z 64.0, A 0, B 90, C 0} C_DIS
$OUT[1] = TRUE
WAIT SEC 0.8
LIN {X -60.0, Y -60.0, Z 64.0, A 0, B 90, C 0} C_DIS
LIN {X -60.0, Y -60.0, Z 64.0, A 0, B 90, C 0} C_DIS
LIN {X -14.4, Y -60.0, Z 64.0, A 0, B 90, C 0} C_DIS
LIN {X 60.0, Y -60.0, Z 64.0, A 0, B 90, C 0} C_DIS
LIN {X 60.0, Y -14.4, Z 64.0, A 0, B 90, C 0} C_DIS
LIN {X 60.0, Y 60.0, Z 64.0, A 0, B 90, C 0} C_DIS
LIN {X 14.4, Y 60.0, Z 64.0, A 0, B 90, C 0} C_DIS
LIN {X -60.0, Y 60.0, Z 64.0, A 0, B 90, C 0} C_DIS
LIN {X -60.0, Y 14.4, Z 64.0, A 0, B 90, C 0} C_DIS
LIN {X -60.0, Y -56.5, Z 64.0, A 0, B 90, C 0} C_DIS
$OUT[1] = FALSE

; END LAYER 31
LIN {X -60.0, Y -60.0, Z 64.0, A 0, B 90, C 0} C_DIS
WAIT SEC 3
LIN {X -60.0, Y -60.0, Z 66.0, A 0, B 90, C 0} C_DIS
$OUT[1] = TRUE
WAIT SEC 0.8
LIN {X -60.0, Y -60.0, Z 66.0, A 0, B 90, C 0} C_DIS
LIN {X -60.0, Y -60.0, Z 66.0, A 0, B 90, C 0} C_DIS
LIN {X -16.8, Y -60.0, Z 66.0, A 0, B 90, C 0} C_DIS
LIN {X 60.0, Y -60.0, Z 66.0, A 0, B 90, C 0} C_DIS
LIN {X 60.0, Y -16.8, Z 66.0, A 0, B 90, C 0} C_DIS
LIN {X 60.0, Y 60.0, Z 66.0, A 0, B 90, C 0} C_DIS
LIN {X 16.8, Y 60.0, Z 66.0, A 0, B 90, C 0} C_DIS
LIN {X -60.0, Y 60.0, Z 66.0, A 0, B 90, C 0} C_DIS
LIN {X -60.0, Y 16.8, Z 66.0, A 0, B 90, C 0} C_DIS
LIN {X -60.0, Y -56.5, Z 66.0, A 0, B 90, C 0} C_DIS
$OUT[1] = FALSE

; END LAYER 32
LIN {X -60.0, Y -60.0, Z 66.0, A 0, B 90, C 0} C_DIS
WAIT SEC 3
LIN {X -60.0, Y -60.0, Z 68.0, A 0, B 90, C 0} C_DIS
$OUT[1] = TRUE
WAIT SEC 0.8
LIN {X -60.0, Y -60.0, Z 68.0, A 0, B 90, C 0} C_DIS
LIN {X -60.0, Y -60.0, Z 68.0, A 0, B 90, C 0} C_DIS
LIN {X -19.2, Y -60.0, Z 68.0, A 0, B 90, C 0} C_DIS
LIN {X 60.0, Y -60.0, Z 68.0, A 0, B 90, C 0} C_DIS
LIN {X 60.0, Y -19.2, Z 68.0, A 0, B 90, C 0} C_DIS
LIN {X 60.0, Y 60.0, Z 68.0, A 0, B 90, C 0} C_DIS
LIN {X 19.2, Y 60.0, Z 68.0, A 0, B 90, C 0} C_DIS
LIN {X -60.0, Y 60.0, Z 68.0, A 0, B 90, C 0} C_DIS
LIN {X -60.0, Y 19.2, Z 68.0, A 0, B 90, C 0} C_DIS
LIN {X -60.0, Y -56.5, Z 68.0, A 0, B 90, C 0} C_DIS
$OUT[1] = FALSE

; END LAYER 33
LIN {X -60.0, Y -60.0, Z 68.0, A 0, B 90, C 0} C_DIS
WAIT SEC 3
LIN {X -60.0, Y -60.0, Z 70.0, A 0, B 90, C 0} C_DIS
$OUT[1] = TRUE
WAIT SEC 0.8
LIN {X -60.0, Y -60.0, Z 70.0, A 0, B 90, C 0} C_DIS
LIN {X -60.0, Y -60.0, Z 70.0, A 0, B 90, C 0} C_DIS
LIN {X -21.6, Y -60.0, Z 70.0, A 0, B 90, C 0} C_DIS
LIN {X 60.0, Y -60.0, Z 70.0, A 0, B 90, C 0} C_DIS
LIN {X 60.0, Y -21.6, Z 70.0, A 0, B 90, C 0} C_DIS
LIN {X 60.0, Y 60.0, Z 70.0, A 0, B 90, C 0} C_DIS
LIN {X 21.6, Y 60.0, Z 70.0, A 0, B 90, C 0} C_DIS
LIN {X -60.0, Y 60.0, Z 70.0, A 0, B 90, C 0} C_DIS
LIN {X -60.0, Y 21.6, Z 70.0, A 0, B 90, C 0} C_DIS
LIN {X -60.0, Y -56.5, Z 70.0, A 0, B 90, C 0} C_DIS
$OUT[1] = FALSE

; END LAYER 34
LIN {X -60.0, Y -60.0, Z 70.0, A 0, B 90, C 0} C_DIS
WAIT SEC 3
LIN {X -60.0, Y -60.0, Z 72.0, A 0, B 90, C 0} C_DIS
$OUT[1] = TRUE
WAIT SEC 0.8
LIN {X -60.0, Y -60.0, Z 72.0, A 0, B 90, C 0} C_DIS
LIN {X -60.0, Y -60.0, Z 72.0, A 0, B 90, C 0} C_DIS
LIN {X -24.0, Y -60.0, Z 72.0, A 0, B 90, C 0} C_DIS
LIN {X 60.0, Y -60.0, Z 72.0, A 0, B 90, C 0} C_DIS
LIN {X 60.0, Y -24.0, Z 72.0, A 0, B 90, C 0} C_DIS
LIN {X 60.0, Y 60.0, Z 72.0, A 0, B 90, C 0} C_DIS
LIN {X 24.0, Y 60.0, Z 72.0, A 0, B 90, C 0} C_DIS
LIN {X -60.0, Y 60.0, Z 72.0, A 0, B 90, C 0} C_DIS
LIN {X -60.0, Y 24.0, Z 72.0, A 0, B 90, C 0} C_DIS
LIN {X -60.0, Y -56.5, Z 72.0, A 0, B 90, C 0} C_DIS
$OUT[1] = FALSE

; END LAYER 35
LIN {X -60.0, Y -60.0, Z 72.0, A 0, B 90, C 0} C_DIS
WAIT SEC 3
LIN {X -60.0, Y -60.0, Z 74.0, A 0, B 90, C 0} C_DIS
$OUT[1] = TRUE
WAIT SEC 0.8
LIN {X -60.0, Y -60.0, Z 74.0, A 0, B 90, C 0} C_DIS
LIN {X -60.0, Y -60.0, Z 74.0, A 0, B 90, C 0} C_DIS
LIN {X -26.4, Y -60.0, Z 74.0, A 0, B 90, C 0} C_DIS
LIN {X 60.0, Y -60.0, Z 74.0, A 0, B 90, C 0} C_DIS
LIN {X 60.0, Y -26.4, Z 74.0, A 0, B 90, C 0} C_DIS
LIN {X 60.0, Y 60.0, Z 74.0, A 0, B 90, C 0} C_DIS
LIN {X 26.4, Y 60.0, Z 74.0, A 0, B 90, C 0} C_DIS
LIN {X -60.0, Y 60.0, Z 74.0, A 0, B 90, C 0} C_DIS
LIN {X -60.0, Y 26.4, Z 74.0, A 0, B 90, C 0} C_DIS
LIN {X -60.0, Y -56.5, Z 74.0, A 0, B 90, C 0} C_DIS
$OUT[1] = FALSE

; END LAYER 36
LIN {X -60.0, Y -60.0, Z 74.0, A 0, B 90, C 0} C_DIS
WAIT SEC 3
LIN {X -60.0, Y -60.0, Z 76.0, A 0, B 90, C 0} C_DIS
$OUT[1] = TRUE
WAIT SEC 0.8
LIN {X -60.0, Y -60.0, Z 76.0, A 0, B 90, C 0} C_DIS
LIN {X -60.0, Y -60.0, Z 76.0, A 0, B 90, C 0} C_DIS
LIN {X -28.8, Y -60.0, Z 76.0, A 0, B 90, C 0} C_DIS
LIN {X 60.0, Y -60.0, Z 76.0, A 0, B 90, C 0} C_DIS
LIN {X 60.0, Y -28.8, Z 76.0, A 0, B 90, C 0} C_DIS
LIN {X 60.0, Y 60.0, Z 76.0, A 0, B 90, C 0} C_DIS
LIN {X 28.8, Y 60.0, Z 76.0, A 0, B 90, C 0} C_DIS
LIN {X -60.0, Y 60.0, Z 76.0, A 0, B 90, C 0} C_DIS
LIN {X -60.0, Y 28.8, Z 76.0, A 0, B 90, C 0} C_DIS
LIN {X -60.0, Y -56.5, Z 76.0, A 0, B 90, C 0} C_DIS
$OUT[1] = FALSE

; END LAYER 37
LIN {X -60.0, Y -60.0, Z 76.0, A 0, B 90, C 0} C_DIS
WAIT SEC 3
LIN {X -60.0, Y -60.0, Z 78.0, A 0, B 90, C 0} C_DIS
$OUT[1] = TRUE
WAIT SEC 0.8
LIN {X -60.0, Y -60.0, Z 78.0, A 0, B 90, C 0} C_DIS
LIN {X -60.0, Y -60.0, Z 78.0, A 0, B 90, C 0} C_DIS
LIN {X -31.2, Y -60.0, Z 78.0, A 0, B 90, C 0} C_DIS
LIN {X 60.0, Y -60.0, Z 78.0, A 0, B 90, C 0} C_DIS
LIN {X 60.0, Y -31.2, Z 78.0, A 0, B 90, C 0} C_DIS
LIN {X 60.0, Y 60.0, Z 78.0, A 0, B 90, C 0} C_DIS
LIN {X 31.2, Y 60.0, Z 78.0, A 0, B 90, C 0} C_DIS
LIN {X -60.0, Y 60.0, Z 78.0, A 0, B 90, C 0} C_DIS
LIN {X -60.0, Y 31.2, Z 78.0, A 0, B 90, C 0} C_DIS
LIN {X -60.0, Y -56.5, Z 78.0, A 0, B 90, C 0} C_DIS
$OUT[1] = FALSE

; END LAYER 38
LIN {X -60.0, Y -60.0, Z 78.0, A 0, B 90, C 0} C_DIS
WAIT SEC 3
LIN {X -60.0, Y -60.0, Z 80.0, A 0, B 90, C 0} C_DIS
$OUT[1] = TRUE
WAIT SEC 0.8
LIN {X -60.0, Y -60.0, Z 80.0, A 0, B 90, C 0} C_DIS
LIN {X -60.0, Y -60.0, Z 80.0, A 0, B 90, C 0} C_DIS
LIN {X -33.6, Y -60.0, Z 80.0, A 0, B 90, C 0} C_DIS
LIN {X 60.0, Y -60.0, Z 80.0, A 0, B 90, C 0} C_DIS
LIN {X 60.0, Y -33.6, Z 80.0, A 0, B 90, C 0} C_DIS
LIN {X 60.0, Y 60.0, Z 80.0, A 0, B 90, C 0} C_DIS
LIN {X 33.6, Y 60.0, Z 80.0, A 0, B 90, C 0} C_DIS
LIN {X -60.0, Y 60.0, Z 80.0, A 0, B 90, C 0} C_DIS
LIN {X -60.0, Y 33.6, Z 80.0, A 0, B 90, C 0} C_DIS
LIN {X -60.0, Y -56.5, Z 80.0, A 0, B 90, C 0} C_DIS
$OUT[1] = FALSE

; END LAYER 39
LIN {X -60.0, Y -60.0, Z 80.0, A 0, B 90, C 0} C_DIS
WAIT SEC 3
LIN {X -60.0, Y -60.0, Z 82.0, A 0, B 90, C 0} C_DIS
$OUT[1] = TRUE
WAIT SEC 0.8
LIN {X -60.0, Y -60.0, Z 82.0, A 0, B 90, C 0} C_DIS
LIN {X -60.0, Y -60.0, Z 82.0, A 0, B 90, C 0} C_DIS
LIN {X -36.0, Y -60.0, Z 82.0, A 0, B 90, C 0} C_DIS
LIN {X 60.0, Y -60.0, Z 82.0, A 0, B 90, C 0} C_DIS
LIN {X 60.0, Y -36.0, Z 82.0, A 0, B 90, C 0} C_DIS
LIN {X 60.0, Y 60.0, Z 82.0, A 0, B 90, C 0} C_DIS
LIN {X 36.0, Y 60.0, Z 82.0, A 0, B 90, C 0} C_DIS
LIN {X -60.0, Y 60.0, Z 82.0, A 0, B 90, C 0} C_DIS
LIN {X -60.0, Y 36.0, Z 82.0, A 0, B 90, C 0} C_DIS
LIN {X -60.0, Y -56.5, Z 82.0, A 0, B 90, C 0} C_DIS
$OUT[1] = FALSE

; END LAYER 40
LIN {X -60.0, Y -60.0, Z 82.0, A 0, B 90, C 0} C_DIS
WAIT SEC 3
LIN {X -60.0, Y -60.0, Z 84.0, A 0, B 90, C 0} C_DIS
$OUT[1] = TRUE
WAIT SEC 0.8
LIN {X -60.0, Y -60.0, Z 84.0, A 0, B 90, C 0} C_DIS
LIN {X -60.0, Y -60.0, Z 84.0, A 0, B 90, C 0} C_DIS
LIN {X -38.4, Y -60.0, Z 84.0, A 0, B 90, C 0} C_DIS
LIN {X 60.0, Y -60.0, Z 84.0, A 0, B 90, C 0} C_DIS
LIN {X 60.0, Y -38.4, Z 84.0, A 0, B 90, C 0} C_DIS
LIN {X 60.0, Y 60.0, Z 84.0, A 0, B 90, C 0} C_DIS
LIN {X 38.4, Y 60.0, Z 84.0, A 0, B 90, C 0} C_DIS
LIN {X -60.0, Y 60.0, Z 84.0, A 0, B 90, C 0} C_DIS
LIN {X -60.0, Y 38.4, Z 84.0, A 0, B 90, C 0} C_DIS
LIN {X -60.0, Y -56.5, Z 84.0, A 0, B 90, C 0} C_DIS
$OUT[1] = FALSE

; END LAYER 41
LIN {X -60.0, Y -60.0, Z 84.0, A 0, B 90, C 0} C_DIS
WAIT SEC 3
LIN {X -60.0, Y -60.0, Z 86.0, A 0, B 90, C 0} C_DIS
$OUT[1] = TRUE
WAIT SEC 0.8
LIN {X -60.0, Y -60.0, Z 86.0, A 0, B 90, C 0} C_DIS
LIN {X -60.0, Y -60.0, Z 86.0, A 0, B 90, C 0} C_DIS
LIN {X -40.8, Y -60.0, Z 86.0, A 0, B 90, C 0} C_DIS
LIN {X 60.0, Y -60.0, Z 86.0, A 0, B 90, C 0} C_DIS
LIN {X 60.0, Y -40.8, Z 86.0, A 0, B 90, C 0} C_DIS
LIN {X 60.0, Y 60.0, Z 86.0, A 0, B 90, C 0} C_DIS
LIN {X 40.8, Y 60.0, Z 86.0, A 0, B 90, C 0} C_DIS
LIN {X -60.0, Y 60.0, Z 86.0, A 0, B 90, C 0} C_DIS
LIN {X -60.0, Y 40.8, Z 86.0, A 0, B 90, C 0} C_DIS
LIN {X -60.0, Y -56.5, Z 86.0, A 0, B 90, C 0} C_DIS
$OUT[1] = FALSE

; END LAYER 42
LIN {X -60.0, Y -60.0, Z 86.0, A 0, B 90, C 0} C_DIS
WAIT SEC 3
LIN {X -60.0, Y -60.0, Z 88.0, A 0, B 90, C 0} C_DIS
$OUT[1] = TRUE
WAIT SEC 0.8
LIN {X -60.0, Y -60.0, Z 88.0, A 0, B 90, C 0} C_DIS
LIN {X -60.0, Y -60.0, Z 88.0, A 0, B 90, C 0} C_DIS
LIN {X -43.2, Y -60.0, Z 88.0, A 0, B 90, C 0} C_DIS
LIN {X 60.0, Y -60.0, Z 88.0, A 0, B 90, C 0} C_DIS
LIN {X 60.0, Y -43.2, Z 88.0, A 0, B 90, C 0} C_DIS
LIN {X 60.0, Y 60.0, Z 88.0, A 0, B 90, C 0} C_DIS
LIN {X 43.2, Y 60.0, Z 88.0, A 0, B 90, C 0} C_DIS
LIN {X -60.0, Y 60.0, Z 88.0, A 0, B 90, C 0} C_DIS
LIN {X -60.0, Y 43.2, Z 88.0, A 0, B 90, C 0} C_DIS
LIN {X -60.0, Y -56.5, Z 88.0, A 0, B 90, C 0} C_DIS
$OUT[1] = FALSE

; END LAYER 43
LIN {X -60.0, Y -60.0, Z 88.0, A 0, B 90, C 0} C_DIS
WAIT SEC 3
LIN {X -60.0, Y -60.0, Z 90.0, A 0, B 90, C 0} C_DIS
$OUT[1] = TRUE
WAIT SEC 0.8
LIN {X -60.0, Y -60.0, Z 90.0, A 0, B 90, C 0} C_DIS
LIN {X -60.0, Y -60.0, Z 90.0, A 0, B 90, C 0} C_DIS
LIN {X -45.6, Y -60.0, Z 90.0, A 0, B 90, C 0} C_DIS
LIN {X 60.0, Y -60.0, Z 90.0, A 0, B 90, C 0} C_DIS
LIN {X 60.0, Y -45.6, Z 90.0, A 0, B 90, C 0} C_DIS
LIN {X 60.0, Y 60.0, Z 90.0, A 0, B 90, C 0} C_DIS
LIN {X 45.6, Y 60.0, Z 90.0, A 0, B 90, C 0} C_DIS
LIN {X -60.0, Y 60.0, Z 90.0, A 0, B 90, C 0} C_DIS
LIN {X -60.0, Y 45.6, Z 90.0, A 0, B 90, C 0} C_DIS
LIN {X -60.0, Y -56.5, Z 90.0, A 0, B 90, C 0} C_DIS
$OUT[1] = FALSE

; END LAYER 44
LIN {X -60.0, Y -60.0, Z 90.0, A 0, B 90, C 0} C_DIS
WAIT SEC 3
LIN {X -60.0, Y -60.0, Z 92.0, A 0, B 90, C 0} C_DIS
$OUT[1] = TRUE
WAIT SEC 0.8
LIN {X -60.0, Y -60.0, Z 92.0, A 0, B 90, C 0} C_DIS
LIN {X -60.0, Y -60.0, Z 92.0, A 0, B 90, C 0} C_DIS
LIN {X -48.0, Y -60.0, Z 92.0, A 0, B 90, C 0} C_DIS
LIN {X 60.0, Y -60.0, Z 92.0, A 0, B 90, C 0} C_DIS
LIN {X 60.0, Y -48.0, Z 92.0, A 0, B 90, C 0} C_DIS
LIN {X 60.0, Y 60.0, Z 92.0, A 0, B 90, C 0} C_DIS
LIN {X 48.0, Y 60.0, Z 92.0, A 0, B 90, C 0} C_DIS
LIN {X -60.0, Y 60.0, Z 92.0, A 0, B 90, C 0} C_DIS
LIN {X -60.0, Y 48.0, Z 92.0, A 0, B 90, C 0} C_DIS
LIN {X -60.0, Y -56.5, Z 92.0, A 0, B 90, C 0} C_DIS
$OUT[1] = FALSE

; END LAYER 45
LIN {X -60.0, Y -60.0, Z 92.0, A 0, B 90, C 0} C_DIS
WAIT SEC 3
LIN {X -60.0, Y -60.0, Z 94.0, A 0, B 90, C 0} C_DIS
$OUT[1] = TRUE
WAIT SEC 0.8
LIN {X -60.0, Y -60.0, Z 94.0, A 0, B 90, C 0} C_DIS
LIN {X -60.0, Y -60.0, Z 94.0, A 0, B 90, C 0} C_DIS
LIN {X -50.4, Y -60.0, Z 94.0, A 0, B 90, C 0} C_DIS
LIN {X 60.0, Y -60.0, Z 94.0, A 0, B 90, C 0} C_DIS
LIN {X 60.0, Y -50.4, Z 94.0, A 0, B 90, C 0} C_DIS
LIN {X 60.0, Y 60.0, Z 94.0, A 0, B 90, C 0} C_DIS
LIN {X 50.4, Y 60.0, Z 94.0, A 0, B 90, C 0} C_DIS
LIN {X -60.0, Y 60.0, Z 94.0, A 0, B 90, C 0} C_DIS
LIN {X -60.0, Y 50.4, Z 94.0, A 0, B 90, C 0} C_DIS
LIN {X -60.0, Y -56.5, Z 94.0, A 0, B 90, C 0} C_DIS
$OUT[1] = FALSE

; END LAYER 46
LIN {X -60.0, Y -60.0, Z 94.0, A 0, B 90, C 0} C_DIS
WAIT SEC 3
LIN {X -60.0, Y -60.0, Z 96.0, A 0, B 90, C 0} C_DIS
$OUT[1] = TRUE
WAIT SEC 0.8
LIN {X -60.0, Y -60.0, Z 96.0, A 0, B 90, C 0} C_DIS
LIN {X -60.0, Y -60.0, Z 96.0, A 0, B 90, C 0} C_DIS
LIN {X -52.8, Y -60.0, Z 96.0, A 0, B 90, C 0} C_DIS
LIN {X 60.0, Y -60.0, Z 96.0, A 0, B 90, C 0} C_DIS
LIN {X 60.0, Y -52.8, Z 96.0, A 0, B 90, C 0} C_DIS
LIN {X 60.0, Y 60.0, Z 96.0, A 0, B 90, C 0} C_DIS
LIN {X 52.8, Y 60.0, Z 96.0, A 0, B 90, C 0} C_DIS
LIN {X -60.0, Y 60.0, Z 96.0, A 0, B 90, C 0} C_DIS
LIN {X -60.0, Y 52.8, Z 96.0, A 0, B 90, C 0} C_DIS
LIN {X -60.0, Y -56.5, Z 96.0, A 0, B 90, C 0} C_DIS
$OUT[1] = FALSE

; END LAYER 47
LIN {X -60.0, Y -60.0, Z 96.0, A 0, B 90, C 0} C_DIS
WAIT SEC 3
LIN {X -60.0, Y -60.0, Z 98.0, A 0, B 90, C 0} C_DIS
$OUT[1] = TRUE
WAIT SEC 0.8
LIN {X -60.0, Y -60.0, Z 98.0, A 0, B 90, C 0} C_DIS
LIN {X -60.0, Y -60.0, Z 98.0, A 0, B 90, C 0} C_DIS
LIN {X -55.2, Y -60.0, Z 98.0, A 0, B 90, C 0} C_DIS
LIN {X 60.0, Y -60.0, Z 98.0, A 0, B 90, C 0} C_DIS
LIN {X 60.0, Y -55.2, Z 98.0, A 0, B 90, C 0} C_DIS
LIN {X 60.0, Y 60.0, Z 98.0, A 0, B 90, C 0} C_DIS
LIN {X 55.2, Y 60.0, Z 98.0, A 0, B 90, C 0} C_DIS
LIN {X -60.0, Y 60.0, Z 98.0, A 0, B 90, C 0} C_DIS
LIN {X -60.0, Y 55.2, Z 98.0, A 0, B 90, C 0} C_DIS
LIN {X -60.0, Y -56.5, Z 98.0, A 0, B 90, C 0} C_DIS
$OUT[1] = FALSE

; END LAYER 48
LIN {X -60.0, Y -60.0, Z 98.0, A 0, B 90, C 0} C_DIS
WAIT SEC 3
LIN {X -60.0, Y -60.0, Z 100.0, A 0, B 90, C 0} C_DIS
$OUT[1] = TRUE
WAIT SEC 0.8
LIN {X -60.0, Y -60.0, Z 100.0, A 0, B 90, C 0} C_DIS
LIN {X -60.0, Y -60.0, Z 100.0, A 0, B 90, C 0} C_DIS
LIN {X -57.6, Y -60.0, Z 100.0, A 0, B 90, C 0} C_DIS
LIN {X 60.0, Y -60.0, Z 100.0, A 0, B 90, C 0} C_DIS
LIN {X 60.0, Y -57.6, Z 100.0, A 0, B 90, C 0} C_DIS
LIN {X 60.0, Y 60.0, Z 100.0, A 0, B 90, C 0} C_DIS
LIN {X 57.6, Y 60.0, Z 100.0, A 0, B 90, C 0} C_DIS
LIN {X -60.0, Y 60.0, Z 100.0, A 0, B 90, C 0} C_DIS
LIN {X -60.0, Y 57.6, Z 100.0, A 0, B 90, C 0} C_DIS
LIN {X -60.0, Y -56.5, Z 100.0, A 0, B 90, C 0} C_DIS
$OUT[1] = FALSE

; END LAYER 49
;END USER CODE
;HOME
;FOLD PTP HOME Vel=10% DEFAULT
$BWDSTART=FALSE
$H_POS=XHOME
PDAT_ACT=PDEFAULT
FDAT_ACT=FHOME
BAS(#PTP_DAT )
BAS (#VEL_PTP,10 )
PTP XHOME
;ENDFOLD
END

--- cuadrado.dat ---
DEFDAT cuadrado()
ENDDAT
